Omron CX-Programmer project NewProject (CX-Programmer 9.73)

# PLC NewPLC1: CP1E N20

## Global symbols (name address type ; comment)
0.01 BOOL  ; pb start
0.03 BOOL  ; RESET
100.01 BOOL  ; LAMP 1
100.02 BOOL  ; LAMP 2
100.03 BOOL  ; LAMP 3
100.04 BOOL  ; LAMP 4
C001 BOOL  ; COUNTER 1
C002 BOOL  ; COUNTER 2
C003 BOOL  ; COUNTER 3
T001 BOOL  ; timer
T002 BOOL  ; TIMER 2
T003 BOOL  ; TIMER 3
T004 BOOL  ; TIMER4

## Program NewProgram1 (cyclic task 0)

### Section Section1

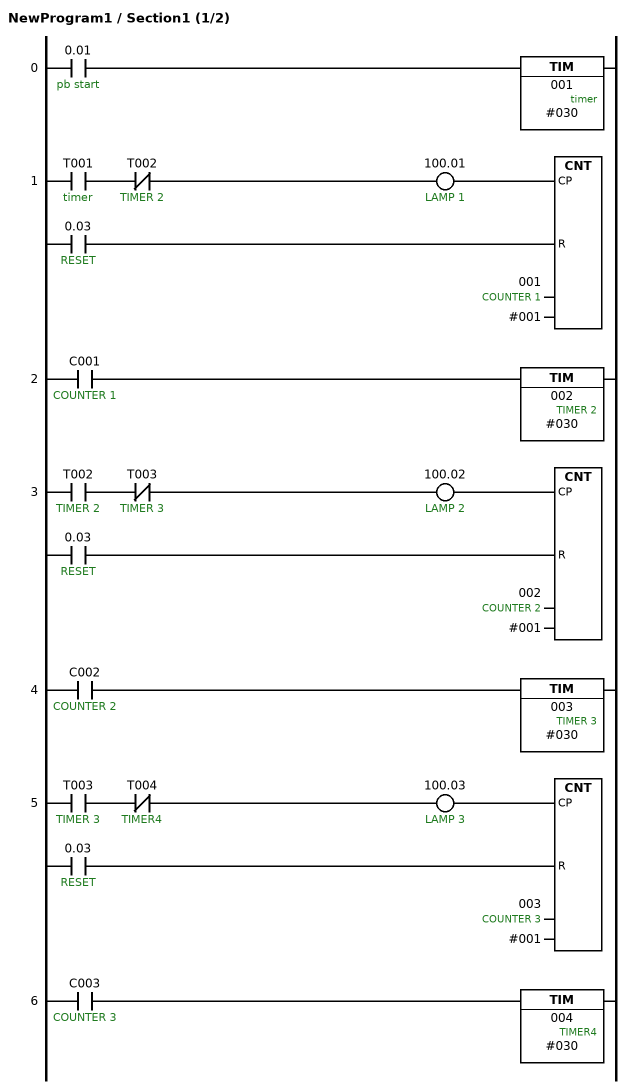
; rung 0
LD 0.01  ; pb start
TIM 001 #030  ; timer
; rung 1
LD T001  ; timer
ANDNOT T002  ; TIMER 2
OUT 100.01  ; LAMP 1
LD 0.03  ; RESET
CNT 001 #001
; rung 2
LD C001  ; COUNTER 1
TIM 002 #030  ; TIMER 2
; rung 3
LD T002  ; TIMER 2
ANDNOT T003  ; TIMER 3
OUT 100.02  ; LAMP 2
LD 0.03  ; RESET
CNT 002 #001
; rung 4
LD C002  ; COUNTER 2
TIM 003 #030  ; TIMER 3
; rung 5
LD T003  ; TIMER 3
ANDNOT T004  ; TIMER4
OUT 100.03  ; LAMP 3
LD 0.03  ; RESET
CNT 003 #001
; rung 6
LD C003  ; COUNTER 3
TIM 004 #030  ; TIMER4

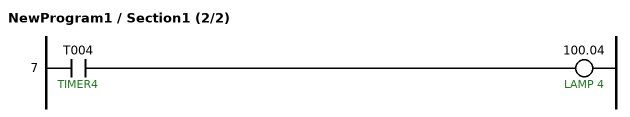
; rung 7
LD T004  ; TIMER4
OUT 100.04  ; LAMP 4

### Section END
; rung 0
END(001)